// Mitsubishi GX Works2 project: label-project   PLC: Q02/Q02H

// global labels: Global1
VAR_GLOBAL
  공급_후_완 AT X0 : BOOL;
  공급_전_완 AT X1 : BOOL;
  드릴_상_완 AT X2 : BOOL;
  드릴_하_완 AT X3 : BOOL;
  송출_후_완 AT X4 : BOOL;
  송출_전_완 AT X5 : BOOL;
  배출_후_완 AT X6 : BOOL;
  배출_전_완 AT X7 : BOOL;
  매거진 AT X8 : BOOL;
  비금속 AT X9 : BOOL;
  금속 AT X0A : BOOL;
  공급_전 AT Y20 : BOOL;
  공급_후 AT Y21 : BOOL;
  드릴_전 AT Y22 : BOOL;
  송출_전 AT Y23 : BOOL;
  송출_후 AT Y24 : BOOL;
  배출_전 AT Y25 : BOOL;
  배출_후 AT Y26 : BOOL;
  컨베이어 AT Y27 : BOOL;
  가공도 AT Y28 : BOOL;
  적색 AT Y29 : BOOL;
  황색 AT Y2A : BOOL;
  녹색 AT Y2B : BOOL;
  PB1 AT X10 : BOOL;
  PB2 AT X11 : BOOL;
  정지 AT X18 : BOOL;
END_VAR

PROGRAM MAIN
VAR
  SELFHOLD_1 : SELFHOLD;
  SELFHOLD_2 : SELFHOLD;
  INTERLOCK_1 : INTERLOCK;
  INTERLOCK_2 : INTERLOCK;
  INTERLOCK_3 : INTERLOCK;
  UPCOUNTER_1 : UPCOUNTER;
  UPCOUNTER_2 : UPCOUNTER;
  DOWN_COUNTER_1 : DOWN_COUNTER;
  REPEATER_1 : REPEATER;
END_VAR
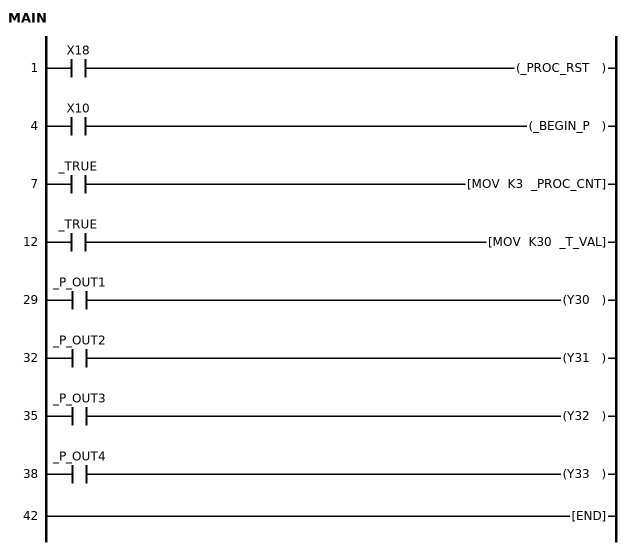
; FB BLK START REPEATER(REPEATER_1)
1     LD      X18
      OUT     _PROC_RST
4     LD      X10
      OUT     _BEGIN_P
7     LD      _TRUE
      MOV     K3 _PROC_CNT
12    LD      _TRUE
      MOV     K30 _T_VAL
; FB START
; FB_NAME REPEATER
; INSTANCE_NAME REPEATER_1
; FB IN_B:PROC_RST
; FB OUT_P_OUT1:B
; FB IN_B:BEGIN_P
; FB OUT_P_OUT2:B
; FB IN_W:PROC_CNT
; FB OUT_P_OUT3:B
; FB IN_W:T_VAL
; FB OUT_P_OUT4:B
; FB END
29    LD      _P_OUT1
      OUT     Y30
32    LD      _P_OUT2
      OUT     Y31
35    LD      _P_OUT3
      OUT     Y32
38    LD      _P_OUT4
      OUT     Y33
; FB BLK END
42    END
END_PROGRAM

FUNCTION_BLOCK SELFHOLD
VAR_INPUT
  IN : BOOL;
  INN2 : BOOL;
END_VAR
VAR_OUTPUT
  OUTT : BOOL;
END_VAR
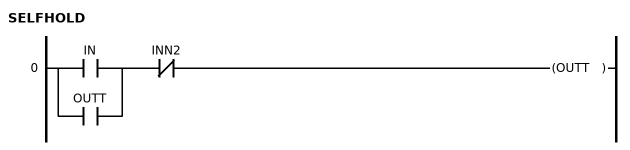
0     LD      IN
      OR      OUTT
      ANI     INN2
      OUT     OUTT
END_FUNCTION_BLOCK

FUNCTION_BLOCK INTERLOCK
VAR_INPUT
  IN1 : BOOL;
  IN2 : BOOL;
END_VAR
VAR_OUTPUT
  OUT1 : BOOL;
  OUT2 : BOOL;
END_VAR
VAR_INPUT
  CUTOFF : BOOL;
END_VAR
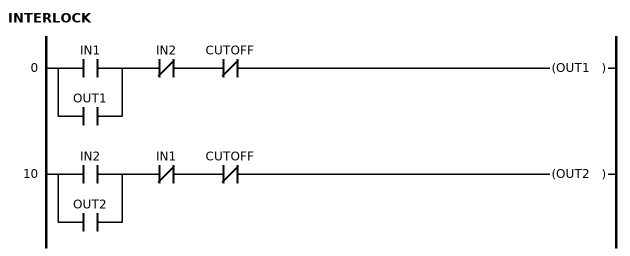
0     LD      IN1
      OR      OUT1
      ANI     IN2
      ANI     CUTOFF
      OUT     OUT1
10    LD      IN2
      OR      OUT2
      ANI     IN1
      ANI     CUTOFF
      OUT     OUT2
END_FUNCTION_BLOCK

FUNCTION_BLOCK UPCOUNTER
VAR_INPUT
  CNT_RESET : BOOL;
  TICK_UP : BOOL;
END_VAR
VAR_OUTPUT
  CNT_DONE : BOOL;
  DATA_REG : INT;
END_VAR
VAR_INPUT
  CNT : INT;
END_VAR
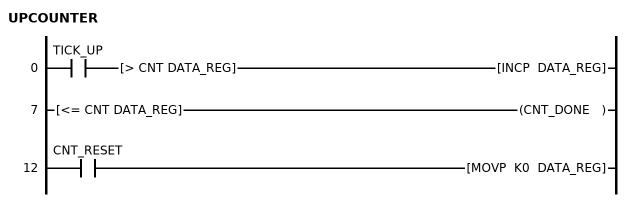
0     LD      TICK_UP
      AND>    CNT DATA_REG
      INCP    DATA_REG
7     LD<=    CNT DATA_REG
      OUT     CNT_DONE
12    LD      CNT_RESET
      MOVP    K0 DATA_REG
END_FUNCTION_BLOCK

FUNCTION_BLOCK DOWN_COUNTER
VAR_INPUT
  CNT_RESET : BOOL;
  TICK_DOWN : BOOL;
  CNT : INT;
END_VAR
VAR_OUTPUT
  CNT_DONE : BOOL;
  CURR_CNT : INT;
END_VAR
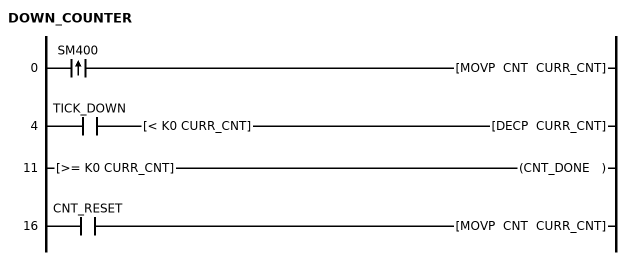
0     LDP     SM400
      MOVP    CNT CURR_CNT
4     LD      TICK_DOWN
      AND<    K0 CURR_CNT
      DECP    CURR_CNT
11    LD>=    K0 CURR_CNT
      OUT     CNT_DONE
16    LD      CNT_RESET
      MOVP    CNT CURR_CNT
END_FUNCTION_BLOCK

FUNCTION_BLOCK REPEATER
VAR_INPUT
  PROC_RST : BOOL;
  BEGIN_P : BOOL;
  PROC_CNT : INT;
END_VAR
VAR_OUTPUT
  P_OUT1 : BOOL;
  P_OUT2 : BOOL;
  P_OUT3 : BOOL;
  P_OUT4 : BOOL;
END_VAR
VAR
  P_STEP : INT;
  TMR_1S : TIMER;
  RUNNING : BOOL;
  REPEAT_CNT : INT;
END_VAR
VAR_INPUT
  T_VAL : INT;
END_VAR
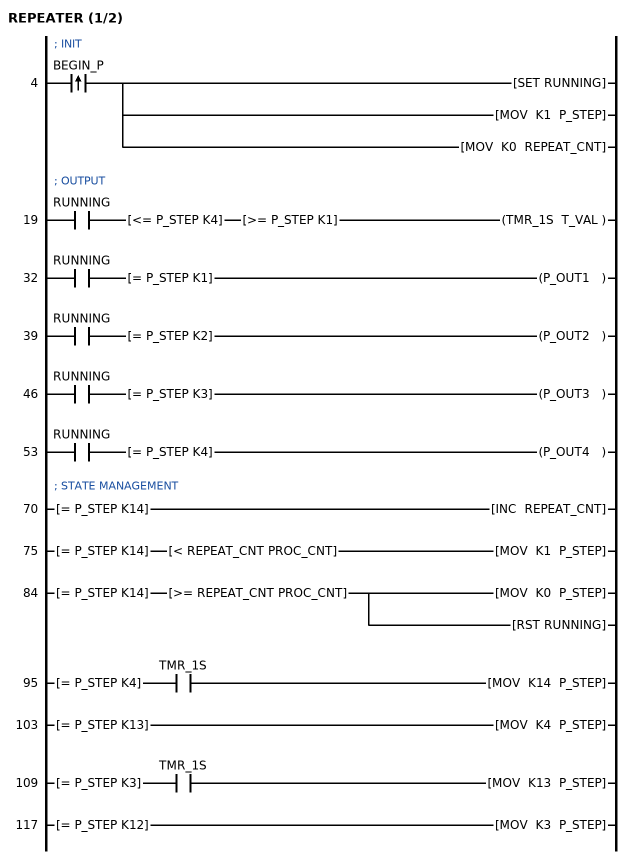
; INIT
4     LDP     BEGIN_P
      SET     RUNNING
      MOV     K1 P_STEP
      MOV     K0 REPEAT_CNT
; OUTPUT
19    LD      RUNNING
      AND<=   P_STEP K4
      AND>=   P_STEP K1
      OUT     TMR_1S T_VAL
32    LD      RUNNING
      AND=    P_STEP K1
      OUT     P_OUT1
39    LD      RUNNING
      AND=    P_STEP K2
      OUT     P_OUT2
46    LD      RUNNING
      AND=    P_STEP K3
      OUT     P_OUT3
53    LD      RUNNING
      AND=    P_STEP K4
      OUT     P_OUT4
; STATE MANAGEMENT
70    LD=     P_STEP K14
      INC     REPEAT_CNT
75    LD=     P_STEP K14
      AND<    REPEAT_CNT PROC_CNT
      MOV     K1 P_STEP
84    LD=     P_STEP K14
      AND>=   REPEAT_CNT PROC_CNT
      MOV     K0 P_STEP
      RST     RUNNING
95    LD=     P_STEP K4
      AND     TMR_1S
      MOV     K14 P_STEP
103   LD=     P_STEP K13
      MOV     K4 P_STEP
109   LD=     P_STEP K3
      AND     TMR_1S
      MOV     K13 P_STEP
117   LD=     P_STEP K12
      MOV     K3 P_STEP
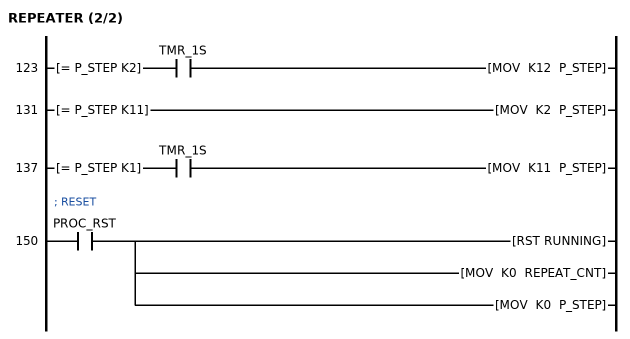
123   LD=     P_STEP K2
      AND     TMR_1S
      MOV     K12 P_STEP
131   LD=     P_STEP K11
      MOV     K2 P_STEP
137   LD=     P_STEP K1
      AND     TMR_1S
      MOV     K11 P_STEP
; RESET
150   LD      PROC_RST
      RST     RUNNING
      MOV     K0 REPEAT_CNT
      MOV     K0 P_STEP
END_FUNCTION_BLOCK
